Fanuc KAREL source: wcnstntpthjt.kl

PROGRAM wcnstntpthjt
%NOLOCKGROUP
VAR
  p : POSITION
  q : POSITION
  i : INTEGER
  r : REAL
BEGIN
  WITH $CNSTNTPTHJT = TRUE MOVE TO p
END wcnstntpthjt
